PROGRAM MAIN
VAR
END_VAR

SAFETY();
GEMMA();
CONVEYOR();
AIS();

(*ST1_HT();*)
(*ST2_ASPIRATION();*)
ST3_ETANCHEITE();
(*ST6_PMAX();*)
(*ST7_SECHAGE();*)
(*ST9_DECHARGEMENT();*)

END_PROGRAM

(* stored: Version 1.1.0.1, ProductVersion 3.1.0.26
   POU MAIN: Id {f2a6ae65-a33b-4129-ab40-ef1a2ef726d5} *)
